{region '#Template'}
	{attribute 'Version' := '5.1.0.0'}
	{attribute 'Tags' := '"LCID": "1031", "Text": "Universal, Control, Presencemonitoring"'}
	{attribute 'Tags' := '"LCID": "1033", "Text": "Universal, Control, Presencemonitoring"'}
	{attribute 'Description' := '"LCID": "1031", "Text": "Präsenzbildung mit Reset"'}
	{attribute 'Description' := '"LCID": "1033", "Text": "Presence-detection with reset-function"'}
{endregion}
FUNCTION_BLOCK FB_BA_PresenceMonitoring
VAR_INPUT
	bPresence				: BOOL;
	bRstDelayTimer			: BOOL;
	bRstManMod				: BOOL;
END_VAR
VAR_INPUT CONSTANT PERSISTENT	
	{attribute 'parameterUnit':= 's'}
	nDlyPrc					: UDINT;			// off-delay presence-detection [s]
END_VAR
	
VAR_OUTPUT
	bRstSwi					: BOOL;
	bPresenceState			: BOOL;	
	bPresenceDelayActive	: BOOL;	
	nCountdownPresence		: UDINT;	
END_VAR
VAR
	tofPrcDetc				: TOF;			
	rtRstDelayTimer			: R_TRIG;		
	rtRstManMod				: R_TRIG;		
	ftPrc					: F_TRIG;	
END_VAR
VAR // added by the converter: edge detectors and wires of the graphical bodies
    _w1, _w2 : ANY;
END_VAR

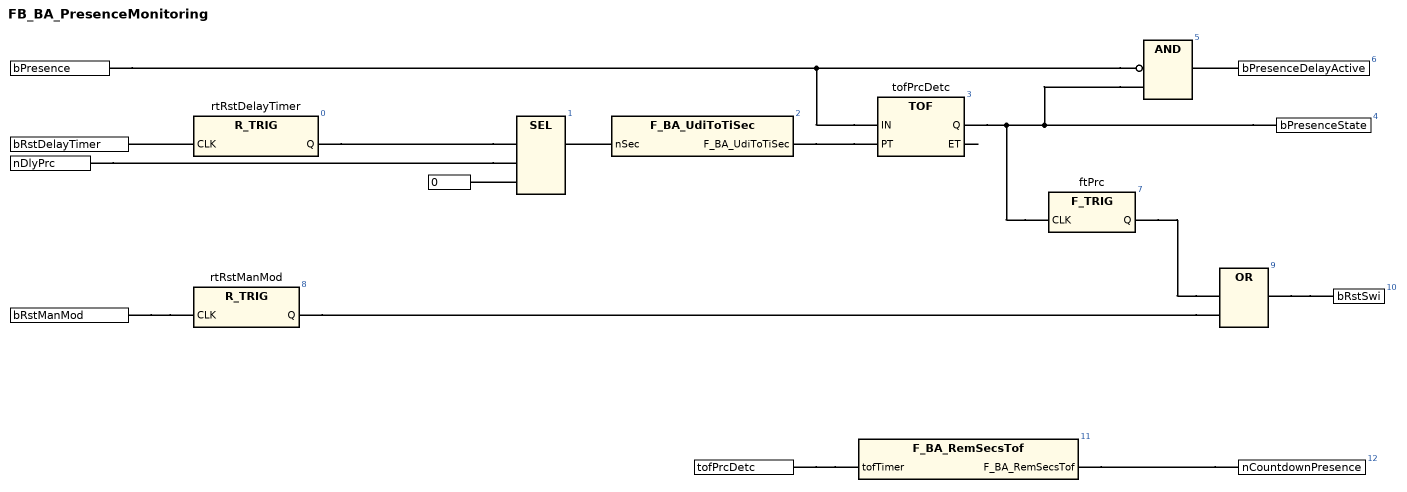
rtRstDelayTimer(CLK := bRstDelayTimer); // R_TRIG
_w1 := F_BA_UdiToTiSec(nSec := SEL(rtRstDelayTimer.Q, nDlyPrc, 0));
tofPrcDetc(IN := bPresence, PT := _w1); // TOF
bPresenceState := tofPrcDetc.Q;
bPresenceDelayActive := NOT bPresence AND tofPrcDetc.Q;
ftPrc(CLK := tofPrcDetc.Q); // F_TRIG
rtRstManMod(CLK := bRstManMod); // R_TRIG
bRstSwi := ftPrc.Q OR rtRstManMod.Q;
_w2 := F_BA_RemSecsTof(tofTimer := tofPrcDetc);
nCountdownPresence := _w2;

METHOD FB_init : BOOL
VAR_INPUT
	bInitRetains : BOOL; // if TRUE, the retain variables are initialized (warm start / cold start)
	bInCopyCode : BOOL;  // if TRUE, the instance afterwards gets moved into the copy code (online change)
END_VAR
nDlyPrc	:= 600;			// off-delay presence-detection [s]
END_METHOD

END_FUNCTION_BLOCK

(* stored: Version 1.1.0.1, ProductVersion 3.1.4024.12
   POU FB_BA_PresenceMonitoring: Id {0bfbed9d-0791-4932-84f3-bf4744c285bb}, SpecialFunc None
   Method FB_init: Id {a6180b6a-7e4e-41ff-ae6e-c4ecea5e39d8} *)
